(* PLC project PLC, Beckhoff Automation GmbH TwinCAT PLC Control 3.5.20.60 *)
(* stored: creationDateTime 2026-07-30T07:42:55.3025569, modificationDateTime 2026-07-30T07:42:55.3065571 *)

TYPE ST_ADS_API_ScadaViewerApp_PLC_Out_Status :

STRUCT

	Mode				:	UINT;												// |1| Hlavní režim stroje
	UserLoggedIn		:	BOOL;												// |2| Hlavní režim stroje
	Order				:	ST_ADS_API_ScadaViewerApp_PLC_Out_Status_Order;		// |3| Informace o zakázce
	Boxes				:	ST_ADS_API_ScadaViewerApp_PLC_Out_Status_Boxes;		// |4| Informace o třídícícíh boxech
	
END_STRUCT

END_TYPE
